{attribute 'linkalways'} 
{attribute 'no_explicit_call' := 'This FB is a CLASS and must be accessed using methods or properties'}
{attribute 'enable_dynamic_creation'}
FUNCTION_BLOCK FINAL MAX_REAL EXTENDS Node
VAR
	in1 : _REAL(0.0);
	in2 : _REAL(0.0);
	out : _REAL(0.0);
END_VAR

METHOD PUBLIC Clone : I_Node
VAR
	pNode : POINTER TO MAX_REAL;
END_VAR
pNode := __NEW(MAX_REAL);
Clone := pNode^;
END_METHOD

METHOD FB_init : BOOL
VAR_INPUT
	bInitRetains : BOOL; // if TRUE, the retain variables are initialized (warm start / cold start)
	bInCopyCode : BOOL;  // if TRUE, the instance afterwards gets moved into the copy code (online change)
END_VAR
AddInput('in1',THIS^.in1);
AddInput('in2',THIS^.in2);
AddOutput('out', THIS^.out);
END_METHOD

METHOD PROTECTED OnExecute
VAR
END_VAR
out.Value := MAX(in1.Value, in2.Value);
END_METHOD

END_FUNCTION_BLOCK

(* stored: Version 1.1.0.1, ProductVersion 3.1.4024.15
   POU MAX_REAL: Id {d6c2508a-2ce7-4787-8ff9-cf06db31f286}, SpecialFunc None
   Folder Constructor: Id {00f1a9c1-db36-497e-9bf6-cbcc3bdef0e4}
   Method Clone: Id {8795474d-f5ba-4f8e-bd23-cee16aa677c3}
   Method FB_init: Id {40522922-026f-43c2-9aae-6388cc3d28f3}
   Method OnExecute: Id {3cba8a24-0528-4e4e-a318-d9066d77f76e} *)
